// TIA Portal project "Comunicao_entre_clps" (V16)

(* hardware
DEVICE "S7-1200 station_1"  S7-1200 Station
   slot 0: "Rack_0"  S7-1200 Rack  Rack  V1.0
   slot 1: "PLC_1"  CPU 1215C DC/DC/DC  6ES7 215-1AG40-0XB0  V4.4
DEVICE "S7-1200 station_2"  S7-1200 Station
   slot 0: "Rack_0"  S7-1200 Rack  Rack  V1.0
   slot 1: "PLC_2"  CPU 1215C DC/DC/DC  6ES7 215-1AG40-0XB0  V4.4
*)

// ===== PLC "PLC_1"  CPU 1215C DC/DC/DC =====

VAR_GLOBAL   // PLC tag table "Default tag table"
   "Clock_Byte" AT %MB50 : Byte;
   "Clock_10Hz" AT %M50.0 : Bool;
   "Clock_5Hz" AT %M50.1 : Bool;
   "Clock_2.5Hz" AT %M50.2 : Bool;
   "Clock_2Hz" AT %M50.3 : Bool;
   "Clock_1.25Hz" AT %M50.4 : Bool;
   "Clock_1Hz" AT %M50.5 : Bool;
   "Clock_0.625Hz" AT %M50.6 : Bool;
   "Clock_0.5Hz" AT %M50.7 : Bool;
   "TESTE_CLP1" AT %MW200 : Int;
   "TESTE2_CLP1" AT %MW202 : Int;
   "TESTE3_CLP1" AT %MW204 : Int;
   "START" AT %M10.0 : Bool;
   "STOP" AT %M10.1 : Bool;
   "MOTOR" AT %M10.2 : Bool;
   "TESTE4_CLP1" AT %MW206 : Int;
END_VAR

DATA_BLOCK "ENVIA"   // DB3
{ S7_Optimized_Access := 'FALSE' }
VERSION : 0.1
   VAR
      VALORPROCESSO : Int;
   END_VAR
BEGIN
END_DATA_BLOCK

DATA_BLOCK "RECEBE"   // DB4
{ S7_Optimized_Access := 'FALSE' }
VERSION : 0.1
   VAR
      RETORNOPROCESSO : Int;
   END_VAR
BEGIN
END_DATA_BLOCK

ORGANIZATION_BLOCK "Main"   // OB1, LAD, ProgramCycle
TITLE = "Main Program Sweep (Cycle)"
{ S7_Optimized_Access := 'TRUE' }
VERSION : 0.1
   VAR_INPUT
      Initial_Call : Bool;   // Initial call of this OB
      Remanence : Bool;   // =True, if remanent data are available
   END_VAR
BEGIN

REGION Network 1
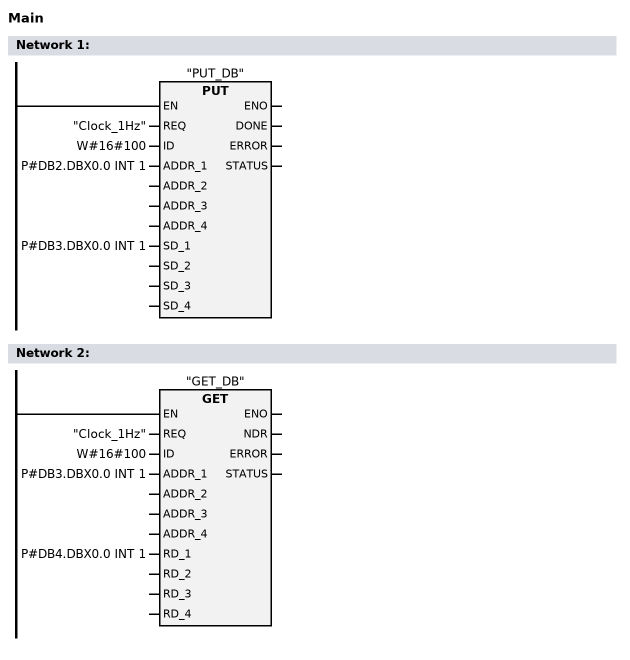
   "PUT_DB"(REQ := "Clock_1Hz", ID := W#16#100, ADDR_1 := P#DB2.DBX0.0 INT 1, SD_1 := P#DB3.DBX0.0 INT 1);   // PUT
END_REGION

REGION Network 2
   "GET_DB"(REQ := "Clock_1Hz", ID := W#16#100, ADDR_1 := P#DB3.DBX0.0 INT 1, RD_1 := P#DB4.DBX0.0 INT 1);   // GET
END_REGION
END_ORGANIZATION_BLOCK

// ===== PLC "PLC_2"  CPU 1215C DC/DC/DC =====

VAR_GLOBAL   // PLC tag table "Default tag table"
   "Clock_Byte" AT %MB50 : Byte;
   "Clock_10Hz" AT %M50.0 : Bool;
   "Clock_5Hz" AT %M50.1 : Bool;
   "Clock_2.5Hz" AT %M50.2 : Bool;
   "Clock_2Hz" AT %M50.3 : Bool;
   "Clock_1.25Hz" AT %M50.4 : Bool;
   "Clock_1Hz" AT %M50.5 : Bool;
   "Clock_0.625Hz" AT %M50.6 : Bool;
   "Clock_0.5Hz" AT %M50.7 : Bool;
   "TESTE_CLP2" AT %MW100 : Int;
   "TESTE2_CLP2" AT %MW102 : Int;
   "TESTE3_CLP2" AT %MW104 : Int;
   "START" AT %M20.0 : Bool;
   "STOP" AT %M20.1 : Bool;
   "MOTOR" AT %M20.2 : Bool;
   "TESTE4_CLP2" AT %MW106 : Int;
END_VAR

DATA_BLOCK "RECEBE_CLP"   // DB2
{ S7_Optimized_Access := 'FALSE' }
VERSION : 0.1
   VAR
      SETPOINT : Int;
   END_VAR
BEGIN
END_DATA_BLOCK

DATA_BLOCK "LEITURA_CLP"   // DB3
{ S7_Optimized_Access := 'FALSE' }
VERSION : 0.1
   VAR
      ANGULO : Int;
   END_VAR
BEGIN
END_DATA_BLOCK

ORGANIZATION_BLOCK "Main"   // OB1, LAD, ProgramCycle
TITLE = "Main Program Sweep (Cycle)"
{ S7_Optimized_Access := 'TRUE' }
VERSION : 0.1
   VAR_INPUT
      Initial_Call : Bool;   // Initial call of this OB
      Remanence : Bool;   // =True, if remanent data are available
   END_VAR
BEGIN

REGION Network 1
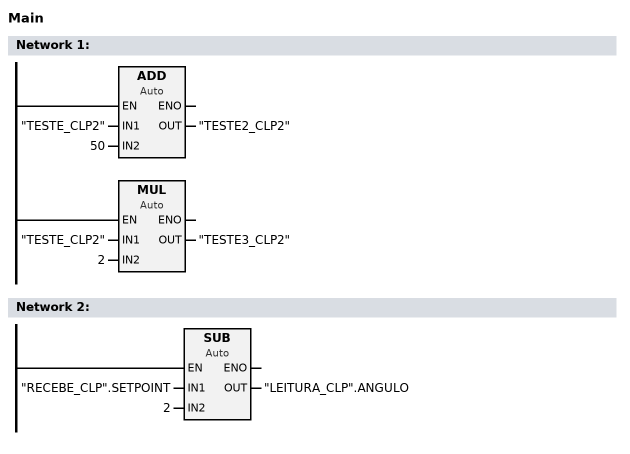
   RUNG wire#powerrail
      Add(in1 := "TESTE_CLP2", in2 := 50, out => "TESTE2_CLP2")
   END_RUNG
   RUNG wire#powerrail
      Mul(in1 := "TESTE_CLP2", in2 := 2, out => "TESTE3_CLP2")
   END_RUNG
   // the same network as SCL:
   "TESTE2_CLP2" := "TESTE_CLP2" + 50;
   "TESTE3_CLP2" := "TESTE_CLP2" * 2;
END_REGION

REGION Network 2
   RUNG wire#powerrail
      Sub(in1 := "RECEBE_CLP".SETPOINT, in2 := 2, out => "LEITURA_CLP".ANGULO)
   END_RUNG
   // the same network as SCL:
   "LEITURA_CLP".ANGULO := "RECEBE_CLP".SETPOINT - 2;
END_REGION
END_ORGANIZATION_BLOCK